FUNCTION_BLOCK VN_model
  (* Version 1.0, 2005-09-21, Goran Cengic, Chalmers *)
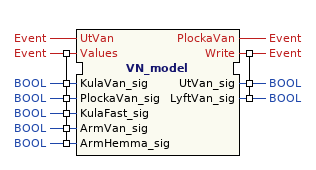
  EVENT_INPUT
    UtVan;
    Values WITH KulaVan_sig, PlockaVan_sig, KulaFast_sig, ArmVan_sig, ArmHemma_sig;
  END_EVENT
  EVENT_OUTPUT
    PlockaVan;
    Write WITH UtVan_sig, LyftVan_sig;
  END_EVENT
  VAR_INPUT
    KulaVan_sig : BOOL;
    PlockaVan_sig : BOOL;
    KulaFast_sig : BOOL;
    ArmVan_sig : BOOL;
    ArmHemma_sig : BOOL;
  END_VAR
  VAR_OUTPUT
    UtVan_sig : BOOL;
    LyftVan_sig : BOOL;
  END_VAR
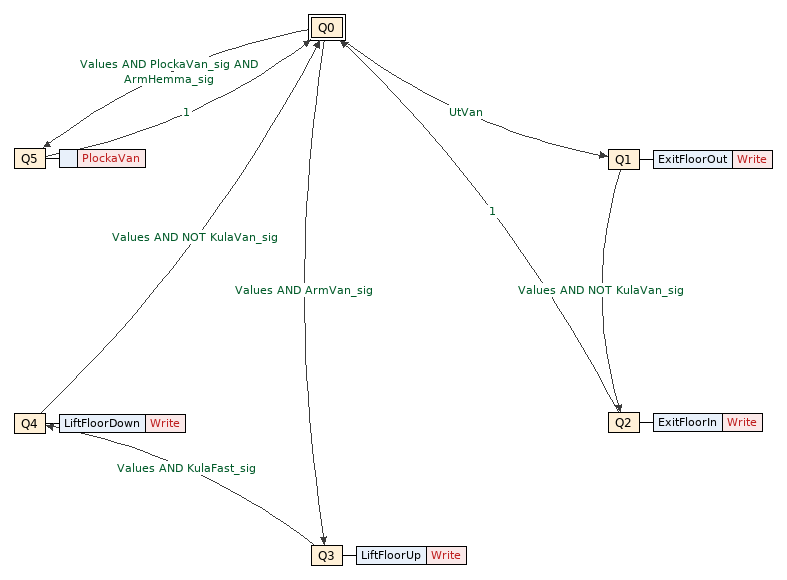
  EC_STATES
    Q0;
    Q1 : ExitFloorOut -> Write;
    Q2 : ExitFloorIn -> Write;
    Q3 : LiftFloorUp -> Write;
    Q4 : LiftFloorDown -> Write;
    Q5 : -> PlockaVan;
  END_STATES
  EC_TRANSITIONS
    Q0 TO Q1 := UtVan;
    Q0 TO Q3 := Values AND ArmVan_sig;
    Q0 TO Q5 := Values AND PlockaVan_sig AND ArmHemma_sig;
    Q1 TO Q2 := Values AND NOT KulaVan_sig;
    Q2 TO Q0 := 1;
    Q3 TO Q4 := Values AND KulaFast_sig;
    Q4 TO Q0 := Values AND NOT KulaVan_sig;
    Q5 TO Q0 := 1;
  END_TRANSITIONS
  ALGORITHM LiftFloorUp IN Java:
		System.out.println("Lifting floor up.");
		LyftVan_sig = true;
  END_ALGORITHM
  ALGORITHM LiftFloorDown IN Java:
		System.out.println("Lifting floor down.");
		LyftVan_sig = false;
  END_ALGORITHM
  ALGORITHM ExitFloorOut IN Java:
		System.out.println("Exiting floor out.");
		UtVan_sig = true;
  END_ALGORITHM
  ALGORITHM ExitFloorIn IN Java:
		System.out.println("Exiting floor in.");
		UtVan_sig = false;
  END_ALGORITHM
END_FUNCTION_BLOCK
(* other elements stored in the file *)
(* ECTransition Source="Q0" Destination="Q5" Condition="Values AND PlockaVan_sig AND ArmHemma_sig AND NOT KulaFast_sig" / *)
